FUNCTION FUN_TimestructToDate : STRING
VAR_INPUT
	stTime : TIMESTRUCT;
END_VAR
VAR
	sTime : STRING;
END_VAR

sTime := SYSTEMTIME_TO_STRING(stTime);
FUN_TimestructToDate := LEFT(sTime,10);

END_FUNCTION

(* stored: Version 1.1.0.1, ProductVersion 3.1.4024.9
   POU FUN_TimestructToDate: Id {405ceef1-ca6e-4aba-96fd-3439f7ffa86b}, SpecialFunc None *)
